Omron CX-Programmer project NewProject (CX-Programmer 9.50)

# PLC NewPLC1: CP1L M

## Global symbols (name address type ; comment)
0.00 BOOL  ; Push ON
0.01 BOOL  ; Push OFF
0.02 BOOL  ; Pompa Keluar
0.03 BOOL  ; Batas Bawah
0.04 BOOL  ; Batas Atas
0.05 BOOL  ; Saklar Suhu
0.06 BOOL  ; Sensor Ultrasonik
100.00 BOOL  ; Pengupas kentang Bold B56 STD Williams Catering Products
100.01 BOOL  ; Sinyal Conveyor Aktif
100.02 BOOL  ; Sinyal Alat Pemotong Kentang aktif
100.03 BOOL  ; Stop Memotong Kentang
100.04 BOOL  ; Mengisi Minyak Goreng
100.05 BOOL  ; Pompa Minyak
100.06 BOOL  ; Pengaduk
100.07 BOOL  ; Pemanas Penggorengan
100.08 BOOL  ; Pengaktif Elevator
100.09 BOOL  ; Motor 2
100.10 BOOL  ; Sinyal Ultra2
100.11 BOOL  ; Motor 1
101.00 BOOL  ; Pengaktif Elevator
101.01 BOOL  ; Motor 2
101.02 BOOL  ; Sinyal Ultra2
101.03 BOOL  ; Motor 1
101.04 BOOL  ; Sinyal Ultra1
101.05 BOOL  ; Alat Pemotong Kentang  Bold R1 Williams Catering Products
101.06 BOOL  ; Alat Conveyor Bekerja
T0000 BOOL  ; Conveyor ON
T0001 BOOL  ; Durasi Conveyor Berjalan ke Pemotong Kentang
T0002 BOOL  ; Durasi Memotong Kentang
T0003 BOOL  ; Durasi Mengaduk
T0004 BOOL  ; Durasi Menggoreng
T0005 BOOL  ; Durasi Motor 2 Bekerja
T0006 BOOL  ; Durasi Motor 1 Bekerja

## Program NewProgram1 (cyclic task 0)

### Section Section1

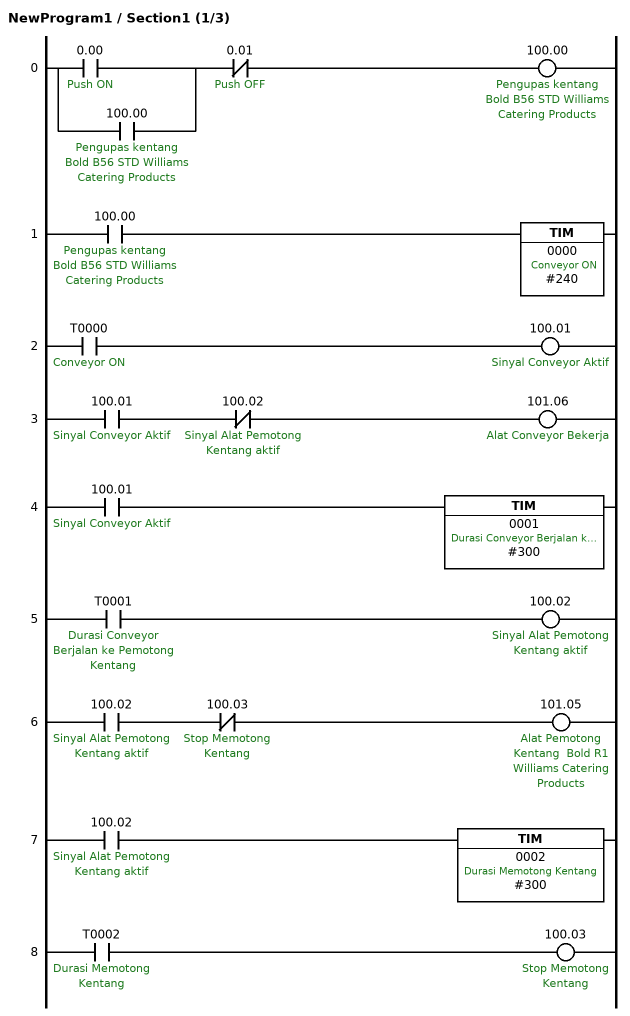
; rung 0
LD 0.00  ; Push ON
OR 100.00  ; Pengupas kentang Bold B56 STD Williams Catering Products
ANDNOT 0.01  ; Push OFF
OUT 100.00  ; Pengupas kentang Bold B56 STD Williams Catering Products
; rung 1
LD 100.00  ; Pengupas kentang Bold B56 STD Williams Catering Products
TIM 0000 #240  ; Conveyor ON
; rung 2
LD T0000  ; Conveyor ON
OUT 100.01  ; Sinyal Conveyor Aktif
; rung 3
LD 100.01  ; Sinyal Conveyor Aktif
ANDNOT 100.02  ; Sinyal Alat Pemotong Kentang aktif
OUT 101.06  ; Alat Conveyor Bekerja
; rung 4
LD 100.01  ; Sinyal Conveyor Aktif
TIM 0001 #300  ; Durasi Conveyor Berjalan ke Pemotong Kentang
; rung 5
LD T0001  ; Durasi Conveyor Berjalan ke Pemotong Kentang
OUT 100.02  ; Sinyal Alat Pemotong Kentang aktif
; rung 6
LD 100.02  ; Sinyal Alat Pemotong Kentang aktif
ANDNOT 100.03  ; Stop Memotong Kentang
OUT 101.05  ; Alat Pemotong Kentang  Bold R1 Williams Catering Products
; rung 7
LD 100.02  ; Sinyal Alat Pemotong Kentang aktif
TIM 0002 #300  ; Durasi Memotong Kentang
; rung 8
LD T0002  ; Durasi Memotong Kentang
OUT 100.03  ; Stop Memotong Kentang

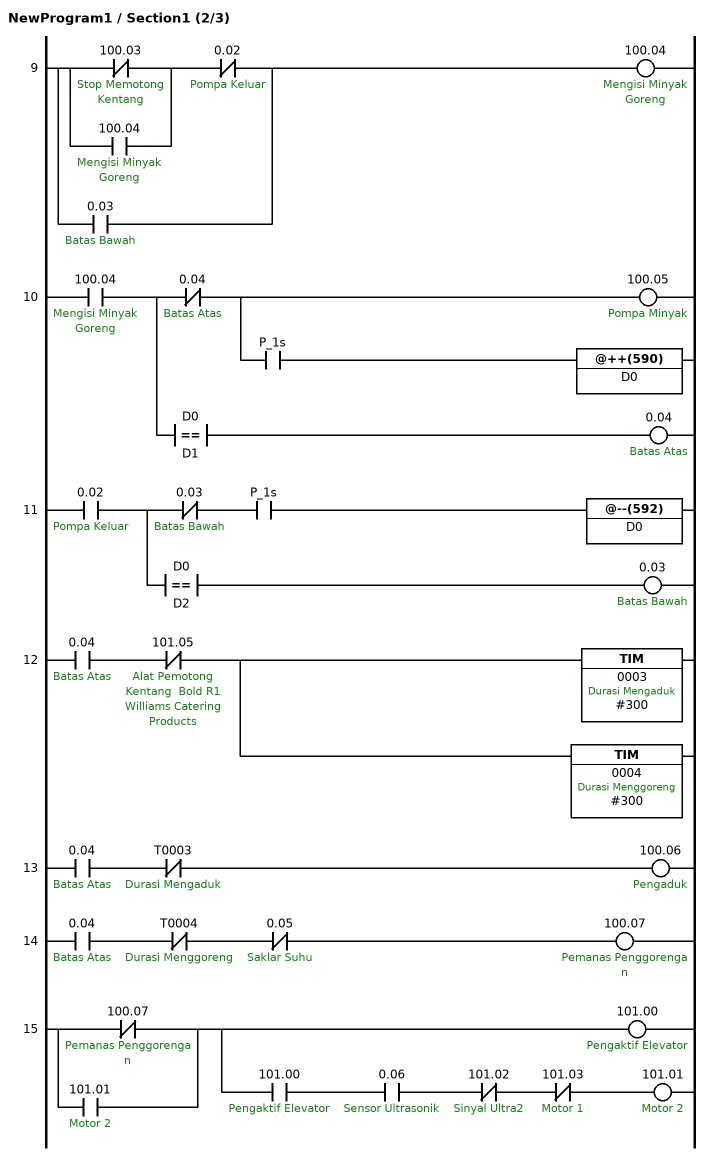
; rung 9
LDNOT 100.03  ; Stop Memotong Kentang
OR 100.04  ; Mengisi Minyak Goreng
ANDNOT 0.02  ; Pompa Keluar
OR 0.03  ; Batas Bawah
OUT 100.04  ; Mengisi Minyak Goreng
; rung 10
LD 100.04  ; Mengisi Minyak Goreng
OUT TR0
ANDNOT 0.04  ; Batas Atas
OUT 100.05  ; Pompa Minyak
AND P_1s
@++(590) D0
LD TR0
AND=(300) D0 D1
OUT 0.04  ; Batas Atas
; rung 11
LD 0.02  ; Pompa Keluar
OUT TR0
ANDNOT 0.03  ; Batas Bawah
AND P_1s
@--(592) D0
LD TR0
AND=(300) D0 D2
OUT 0.03  ; Batas Bawah
; rung 12
LD 0.04  ; Batas Atas
ANDNOT 101.05  ; Alat Pemotong Kentang  Bold R1 Williams Catering Products
TIM 0003 #300  ; Durasi Mengaduk
TIM 0004 #300  ; Durasi Menggoreng
; rung 13
LD 0.04  ; Batas Atas
ANDNOT T0003  ; Durasi Mengaduk
OUT 100.06  ; Pengaduk
; rung 14
LD 0.04  ; Batas Atas
ANDNOT T0004  ; Durasi Menggoreng
ANDNOT 0.05  ; Saklar Suhu
OUT 100.07  ; Pemanas Penggorengan
; rung 15
LDNOT 100.07  ; Pemanas Penggorengan
OR 101.01  ; Motor 2
OUT 101.00  ; Pengaktif Elevator
AND 101.00  ; Pengaktif Elevator
AND 0.06  ; Sensor Ultrasonik
ANDNOT 101.02  ; Sinyal Ultra2
ANDNOT 101.03  ; Motor 1
OUT 101.01  ; Motor 2

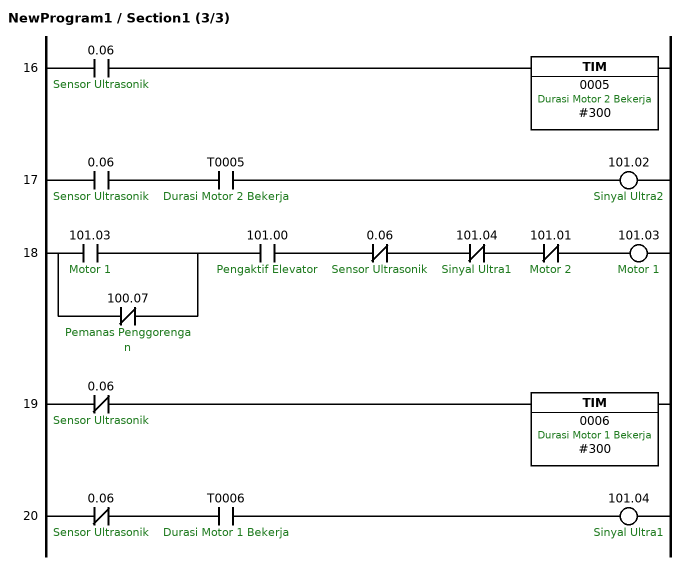
; rung 16
LD 0.06  ; Sensor Ultrasonik
TIM 0005 #300  ; Durasi Motor 2 Bekerja
; rung 17
LD 0.06  ; Sensor Ultrasonik
AND T0005  ; Durasi Motor 2 Bekerja
OUT 101.02  ; Sinyal Ultra2
; rung 18
LD 101.03  ; Motor 1
ORNOT 100.07  ; Pemanas Penggorengan
AND 101.00  ; Pengaktif Elevator
ANDNOT 0.06  ; Sensor Ultrasonik
ANDNOT 101.04  ; Sinyal Ultra1
ANDNOT 101.01  ; Motor 2
OUT 101.03  ; Motor 1
; rung 19
LDNOT 0.06  ; Sensor Ultrasonik
TIM 0006 #300  ; Durasi Motor 1 Bekerja
; rung 20
LDNOT 0.06  ; Sensor Ultrasonik
AND T0006  ; Durasi Motor 1 Bekerja
OUT 101.04  ; Sinyal Ultra1

### Section END
; rung 0
END(001)